(* IEC 61131-3 sources: soft-plc/openplc-editor/project, 1 file *)

(* ---- program.st ---- *)
PROGRAM My_First_Program
  VAR
    PB1 AT %IX0.0 : BOOL;
    PB2 AT %IX0.1 : BOOL;
    LAMP AT %QX0.0 : BOOL;
  END_VAR

  LAMP := NOT(PB2) AND (LAMP OR PB1);
END_PROGRAM

CONFIGURATION Config0

  RESOURCE Res0 ON PLC
    TASK task0(INTERVAL := T#20ms,PRIORITY := 0);
    PROGRAM instance0 WITH task0 : My_First_Program;
  END_RESOURCE
END_CONFIGURATION
